{attribute 'no_explicit_call' := 'do not call this POU directly'} 
FUNCTION_BLOCK FB_StringBuilder IMPLEMENTS I_StringBuilder
VAR_INPUT
END_VAR
VAR_OUTPUT
END_VAR
VAR
	pList:			POINTER TO BYTE;
	aList:			POINTER TO POINTER TO STRING(1000):= ADR(pList);
	nLength:		UDINT;
END_VAR

METHOD M_Append : I_StringBuilder
VAR_INPUT
	Value	: STRING(255);
END_VAR
VAR
	nLengthOld:	UDINT:= nLength;
	pOldList: 	POINTER TO BYTE:=pList;;
END_VAR
// First Item
IF pList = 0 THEN
	nLength:= LEN2(ADR(Value));
	pList:= __NEW(BYTE, (nLength));
ELSE
	// new Length
	nLength:= nLength + LEN2(ADR(Value));
	// new pointer
	pList:= __NEW(BYTE, DINT_TO_UDINT(SIZEOF(BYTE) * nLength));
	// restore
	Memcpy(pList,pOldList, SIZEOF(BYTE)*DINT_TO_UDINT(SIZEOF(BYTE) * nLengthOld));
	// delete old
	__DELETE(pOldList);

END_IF
Memcpy((pList + nLengthOld) , ADR(Value), SIZEOF(BYTE)* LEN2(ADR(Value)));
M_Append:= THIS^;
END_METHOD

METHOD PUBLIC M_AppendBool  : I_StringBuilder
VAR_INPUT
	Value:			BOOL;
END_VAR
M_Append(BOOL_TO_STRING(Value));
M_AppendBool:= THIS^;
END_METHOD

METHOD PUBLIC M_AppendInt : I_StringBuilder
VAR_INPUT
	Value	: LINT;
END_VAR
M_Append(LINT_TO_STRING(Value));
M_AppendInt:= THIS^;
END_METHOD

METHOD PUBLIC M_AppendReal : I_StringBuilder
VAR_INPUT
	Value:		LREAL;
	nDecimals:	SINT;
END_VAR
M_Append(LREAL_TO_FMTSTR(Value, nDecimals, TRUE));
M_AppendReal:= THIS^;
END_METHOD

METHOD M_Copy : BOOL
VAR_INPUT
	Value:			ANY;
END_VAR
Memset(Value.pValue, 0, Value.diSize);
Memcpy(Value.pValue, pList, nLength);
END_METHOD

METHOD M_Find : UDINT
VAR_INPUT
	sValue: STRING;
END_VAR
M_Find:= FIND2(pList, adr(sValue));
END_METHOD

METHOD M_Insert : I_StringBuilder
VAR_INPUT
	nPosition:		UDINT;
	Value:			STRING(255);
END_VAR
INSERT2(pData, ADR(Value), pData, nLength, nIndex);
M_Insert:= THIS^;
END_METHOD

METHOD M_Replace : I_StringBuilder
VAR_INPUT
	ValueOld:		STRING;
	ValueNew:		STRING;
END_VAR
FindAndReplace(pList, ADR(ValueOld), ADR(ValueNew), pList, nLength);
M_Replace:= THIS^;
END_METHOD

METHOD M_Reset : I_StringBuilder
__DELETE(pList);
nLength:= 0;
M_Reset:= THIS^;
END_METHOD

END_FUNCTION_BLOCK

(* stored: Version 1.1.0.1
   POU FB_StringBuilder: Id {019c017e-2b82-4b97-aaf7-21192bfab875}, SpecialFunc None
   Method M_Append: Id {7db82bd1-a9eb-4060-8216-5ab95be3d951}
   Method M_AppendBool: Id {bfecdd7b-04e9-4b45-8de6-ce56cee3d775}
   Method M_AppendInt: Id {111c7396-9c3f-42fb-91f0-39c8d5232d3f}
   Method M_AppendReal: Id {2d407a54-01d7-4964-a23b-5eaea946942e}
   Method M_Copy: Id {3548b8eb-f19a-4821-aca6-7a57d9eaf053}
   Method M_Find: Id {79a92e52-0a6b-451a-9c7f-ae52f055d960}
   Method M_Insert: Id {927c5159-aa65-45c4-a091-434197aceab2}
   Method M_Replace: Id {241f6b9e-97e0-4502-960e-f0846a16abf8}
   Method M_Reset: Id {df3bd2f2-c8d9-4da1-a2f9-320a3b463940} *)
